(* IEC 61131-3 sources: learning-path/05_introduction_to_st/exercises/3_extend_tank_functionality/src, 2 files *)

(* ---- tank.st ---- *)
USING Siemens.AxTraining.ControlModules;
NAMESPACE Siemens.AxTraining.EquipmentModules

    FUNCTION_BLOCK Tank

        VAR_INPUT
            cmdFill : BOOL;
            cmdEmpty : BOOL;
        END_VAR
        VAR_OUTPUT
            inletOpen : BOOL;
            outletOpen : BOOL;
        END_VAR
        VAR
            inlet : Valve;
            outlet : Valve;
        END_VAR;

        inlet(cmdOpen := cmdFill,
                cmdClose := NOT cmdFill,
                ctrlOpen => inletOpen);
        outlet(cmdOpen := cmdEmpty,
                cmdClose := NOT cmdEmpty,
                ctrlOpen => outletOpen);

    END_FUNCTION_BLOCK

END_NAMESPACE

(* ---- configuration.st ---- *)
USING Siemens.AxTraining;

    CONFIGURATION PLC_1
        TASK Main(Interval := T#10ms, Priority := 1);
        PROGRAM P1 WITH Main: FluidProgram;

        VAR_GLOBAL
            cmdFillTank : BOOL;
            cmdEmptyTank : BOOL;
            inletOpenTank : BOOL;
            outletOpenTank : BOOL;
        END_VAR
    END_CONFIGURATION
